KUKA KRL program: ThresholdMillDrainage.src, ThresholdMillDrainage.dat

--- ThresholdMillDrainage.src ---
&ACCESS RVO1
&REL 3
DEF ThresholdMillDrainage(rDrainageX:IN)
   ;FOLD DECL
      DECL REAL rDrainageX
      DECL E_ProfileType eProfileType
      DECL POS xAboveTable,xAboveThreshold
      DECL POS xAwayDrainage,xDrainage,xDrainageAngle
      DECL POS xWall[2],xAboveWall[2],xInsideWall[2]
      DECL POS xCutOffset
      DECL INT iCutPathSize[2]
      DECL POS xCutPath[2,60]
      DECL INT iPoint,iCutIdx,iLayer,iWall,iCycle
   ;ENDFOLD (DECL)
   ;FOLD INI

      ;Get data from ProcessData structure
      eProfileType = gstProcessData.eProfileType

      ;Take the right profile data
      SWITCH eProfileType
         CASE #Threshold90
            xDrainage = xThreshold90
         DEFAULT
            HALT
      ENDSWITCH

      ;Drainage X coordinate
      xDrainage.X = rDrainageX

      ;komentarz i redukcja punktow
      xDrainageAngle  = xDrainage:xMillAngleCorrection
      xAwayDrainage = xDrainageAngle:xAwayDrainageOffset
      xAboveThreshold = xAboveThresholdOffset:xDrainageAngle
      xAboveTable = xAboveTableOffset:xDrainageAngle

      ;Profile walls
      xWall[1] = xDrainage
      xWall[2] = xDrainage:xWallOffset

      ;CutPath[] array size
      iCutPathSize[1] = iRoughCutSize*iLayerSize + iFinishCutSize
      iCutPathSize[2] = iRoughCutSize*iLayerSize

      ;Rough milling coordinates
      FOR iWall=1 TO iWallSize STEP 1
         FOR iLayer=1 TO iLayerSize STEP 1
            FOR iPoint=1 TO iRoughCutSize STEP 1
               xCutOffset = xRoughCut[iPoint]
               SWITCH iPoint
                  CASE 1,2
                     ;Cutting depth for first motion
                     xCutOffset.Z = (iLayer-0.5) * (-rLayerStepZ)
                  CASE 3,4
                     ;Cutting depth for second motion
                     xCutOffset.Z = iLayer * (-rLayerStepZ)
                  DEFAULT
                     HALT
               ENDSWITCH
               iCutIdx = iRoughCutSize*(iLayer-1) + iPoint
               xCutPath[iWall,iCutIdx] = xWall[iWall]:xCutOffset:xMillAngleCorrection
            ENDFOR
         ENDFOR
      ENDFOR

      ;Finish milling coordinates
      FOR iPoint=1 TO iFinishCutSize STEP 1
         iCutIdx = iRoughCutSize*iLayerSize + iPoint
         xCutOffset = xFinishCut[iPoint]
         xCutOffset.Z = -1 * rLayerStepZ*iLayerSize
         xCutPath[1,iCutIdx] = xWall[1]:xCutOffset:xMillAngleCorrection
      ENDFOR

      ;xAboveWall[],xInsideWall[]
      FOR iWall=1 TO iWallSize STEP 1
         xAboveWall[iWall] = xCutPath[iWall,1]:xAboveWallOffset
         xInsideWall[iWall] = xWall[iWall]:xInsideWallOffset:xMillAngleCorrection
      ENDFOR

   ;ENDFOLD (INI)

   SetBaseTool(#MillTable,#ThresholdCutter)

   SetVel(#SpindleIdle)
   LIN xAboveTable C_DIS
   LIN xAboveThreshold C_DIS
   LIN xAwayDrainage C_DIS

   ;Profile milling
   SetVel(#SpindleIdle)
   FOR iWall=1 TO iWallSize STEP 1
      ;Cutter above wall
      LIN xAboveWall[iWall]
      ;Drainage milling
      FOR iPoint=1 TO iCutPathSize[iWall] STEP 1
         SetVel(#MillThreshold)
         LIN xCutPath[iWall,iPoint] C_DIS
      ENDFOR
      ;Cutter inside wall
      LIN xInsideWall[iWall]
   ENDFOR
   ;Away from profile
   LIN xAwayDrainage

   SetVel(#SpindleIdle)
   LIN xAboveThreshold C_DIS
   LIN xAboveTable

END

--- ThresholdMillDrainage.dat ---
&ACCESS RVO1
&REL 3
DEFDAT ThresholdMillDrainage

   DECL CONST POS xThreshold90 = {x 0.0,y 83.0,z 5.8,a 0.0,b 0.0,c -105.0}

   DECL CONST POS xAboveTableOffset = {x 0,y 100,z 200,a 0,b 0,c 0}
   DECL CONST POS xAboveThresholdOffset = {x 0,y 50,z 80,a 0,b 0,c 0}
   DECL CONST POS xAwayDrainageOffset = {x 0,y 0,z 10,a 0,b 0,c 0}

   DECL CONST POS xWallOffset = {X 0.0,Y 0.0,Z -26.0,A 0.0,B 0.0,C 0.0}
   DECL CONST POS xMillAngleCorrection = {x 0,y 0,z 0,a -120,b 0,c 0}
   DECL CONST POS xAboveWallOffset = {x 0,y 0,z 2,a 0,b 0,c 0}
   DECL CONST POS xInsideWallOffset = {x 0,y 0,z -2,a 0,b 0,c 0}

   ;Amount of walls
   DECL CONST INT iWallSize = 2
   ;Amount of wall milling layers
   DECL CONST INT iLayerSize = 11
   ;Depth step by layer
   DECL CONST REAL rLayerStepZ = 0.5

   ;Rough cutting
   DECL CONST INT iRoughCutSize = 4
   DECL CONST POS xRoughCut[4]
   xRoughCut[1] = {X  10.0,Y 0.0,Z 0.0,A 0.0,B 0.0,C 0.0}
   xRoughCut[2] = {X -10.0,Y 0.0,Z 0.0,A 0.0,B 0.0,C 0.0}
   xRoughCut[3] = {X -10.0,Y 0.0,Z 0.0,A 0.0,B 0.0,C 0.0}
   xRoughCut[4] = {X  10.0,Y 0.0,Z 0.0,A 0.0,B 0.0,C 0.0}

   DECL CONST INT iFinishCutSize = 6
   DECL CONST POS xFinishCut[6]
   xFinishCut[1] = {X  10.6,Y -0.6,Z 0.0,A 0.0,B 0.0,C 0.0}
   xFinishCut[2] = {X  10.6,Y  0.6,Z 0.0,A 0.0,B 0.0,C 0.0}
   xFinishCut[3] = {X -10.6,Y  0.6,Z 0.0,A 0.0,B 0.0,C 0.0}
   xFinishCut[4] = {X -10.6,Y -0.6,Z 0.0,A 0.0,B 0.0,C 0.0}
   xFinishCut[5] = {X  10.6,Y -0.6,Z 0.0,A 0.0,B 0.0,C 0.0}
   xFinishCut[6] = {X  10.6,Y  0.6,Z 0.0,A 0.0,B 0.0,C 0.0}

ENDDAT
